FUNCTION_BLOCK FB_Robotersteuerung
VAR_INPUT
    bEnable     : BOOL;
    bExecute    : BOOL;

	bSensBand4 	: BOOL;
	bSensEndX : BOOL;
	bSensEndY : BOOL;
	bSensEndZ : BOOL;
	bSensEndG : BOOL;
END_VAR

VAR_OUTPUT
    eState          : eBetriebszustand;
    bBrakeZ         : BOOL;
    bGripperClosed  : BOOL;
END_VAR

VAR_IN_OUT
    axX : Axis_Ref;
    axY : Axis_Ref;
    axZ : Axis_Ref;
	axG : Axis_Ref;
	
	nLagerIndex : INT; 
END_VAR

VAR
    fbAchseX : FB_AchsenRoboter;
    fbAchseY : FB_AchsenRoboter;
    fbAchseZ : FB_AchsenRoboter;
	fbAchseG : FB_AchsenRoboter;
	
    fbWaage 	: FB_Waage_Temp;
    fbThermo	: FB_Thermo_Temp;

	rGzu 	: REAL 	:= 9.5;
	rGauf 	: REAL 	:= 6.5;
	
    bGreifer	: BOOL;
    nState   	: INT;
END_VAR

fbAchseX(
    bEnable := bEnable,
    bExecute := ,
    rPosition := ,
    bSensEndstop := bSensEndX,
    eState => ,
    ax := axX);

fbAchseY(
    bEnable := bEnable,
    bExecute := ,
    rPosition := ,
    bSensEndstop := bSensEndY,
    eState => ,
    ax := axY);

fbAchseZ(
    bEnable := bEnable,
    bExecute := ,
    rPosition := ,
    bSensEndstop := bSensEndZ,
    eState => ,
    ax := axZ);

fbAchseG(
    bEnable := bEnable,
    bExecute := ,
    rPosition := ,
    bSensEndstop := bSensEndG,
    eState => ,
    ax := axG);

fbWaage();
fbThermo();

CASE nState OF

    0: // OFF
        eState := eBetriebszustand.Off;
        bBrakeZ := FALSE;
        bGripperClosed := FALSE;
		nLagerIndex := 1;
        fbAchseG(bExecute := TRUE, rPosition := rGauf, ax := axG);
        IF bEnable THEN
            nState := 10;
        END_IF

    10: // INIT
        eState := eBetriebszustand.Init;
        bBrakeZ := FALSE;
		fbAchseX(bExecute := TRUE, rPosition := GVL_PosKinematic.pXHome, ax := axX);
        fbAchseY(bExecute := TRUE, rPosition := GVL_PosKinematic.pYHome, ax := axY);
		fbAchseZ(bExecute := TRUE, rPosition := GVL_PosKinematic.pZHome, ax := axZ);
        IF fbAchseX.eState = eBetriebszustand.Done AND fbAchseY.eState = eBetriebszustand.Done AND fbAchseZ.eState = eBetriebszustand.Done THEN
			fbAchseX.bExecute := FALSE;
			fbAchseY.bExecute := FALSE;
			fbAchseZ.bExecute := FALSE;
        	nState := 20;
		END_IF
    20: // READY
        eState := eBetriebszustand.Ready;
        IF bBandSens4 THEN
            nState := 30;
        END_IF

    30: // Z-Achse sicherheits Ebene
        bBrakeZ := TRUE;
        fbAchseZ(bExecute := TRUE, rPosition := GVL_PosKinematic.pZoff, ax := axZ);
        IF fbAchseZ.eState = eBetriebszustand.Done THEN
			fbAchseZ.bExecute := FALSE;
            nState := 31;
        END_IF

    31: // XY Abfüllstation
    IF fbAchseZ.rPosition <= GVL_PosKinematic.pZOff  THEN
		bBrakeZ := FALSE;
        fbAchseX(bExecute := TRUE, rPosition := GVL_PosKinematic.pXconv, ax := axX);
        fbAchseY(bExecute := TRUE, rPosition := GVL_PosKinematic.pYconv, ax := axY);
        IF fbAchseX.eState = eBetriebszustand.Done AND fbAchseY.eState = eBetriebszustand.Done THEN
			fbAchseX.bExecute := FALSE;
			fbAchseY.bExecute := FALSE;
            nState := 32;
        END_IF
    END_IF

    32: // Z-Achse Greifenhöhe
	IF fbAchseX.rPosition = GVL_PosKinematic.pXconv AND 
	   fbAchseY.rPosition = GVL_PosKinematic.pYconv THEN
	   bBrakeZ := TRUE;
        fbAchseZ(bExecute := TRUE, rPosition := GVL_PosKinematic.pZconv, ax := axZ);
        IF fbAchseZ.eState = eBetriebszustand.Done THEN
			fbAchseZ.bExecute := FALSE;
            nState := 33;
        END_IF
	END_IF
	
    33: // Greifen
	IF fbAchseZ.rPosition = GVL_PosKinematic.pZconv AND fbAchseZ.bExecute = FALSE THEN
		bBrakeZ := FALSE;
        fbAchseG(bExecute := TRUE, rPosition := rGzu, ax := axG);
        IF fbAchseG.eState = eBetriebszustand.Done THEN
			fbAchseG.bExecute := FALSE;
            bGripperClosed := TRUE;
            nState := 34;
        END_IF
	END_IF
	
    34: // Z-Achse sicherheits Ebene
	IF fbAchseg.rPosition = rGzu THEN
		bBrakeZ := TRUE;
        fbAchseZ(bExecute := TRUE, rPosition := GVL_PosKinematic.pZoff, ax := axZ);
        IF fbAchseZ.eState = eBetriebszustand.Done THEN
			fbAchseZ.bExecute := FALSE;
            bBrakeZ := TRUE;
            nState := 40;
        END_IF
	END_IF
	
    40: // XY Waage
    IF fbAchseZ.rPosition <= GVL_PosKinematic.pZOff  THEN
		bBrakeZ := FALSE;
        fbAchseX(bExecute := TRUE, rPosition := GVL_PosKinematic.pXscale, ax := axX);
        fbAchseY(bExecute := TRUE, rPosition := GVL_PosKinematic.pYscale, ax := axY);
        IF fbAchseX.eState = eBetriebszustand.Done AND fbAchseY.eState = eBetriebszustand.Done THEN
			fbAchseX.bExecute := FALSE;
			fbAchseY.bExecute := FALSE;
            nState := 41;
        END_IF
    END_IF

    41: // Z-Achse Ablegen
	IF fbAchseX.rPosition = GVL_PosKinematic.pXscale AND 
	   fbAchseY.rPosition = GVL_PosKinematic.pYscale THEN
	    bBrakeZ := TRUE;
        fbAchseZ(bExecute := TRUE, rPosition := GVL_PosKinematic.pZscale, ax := axZ);
        IF fbAchseZ.eState = eBetriebszustand.Done THEN
			fbAchseZ.bExecute := FALSE;
            nState := 42;
        END_IF
	END_IF
	
    42: // Greifer öffnen
	IF fbAchseZ.rPosition = GVL_PosKinematic.pZscale THEN
		bBrakeZ := FALSE;
        fbAchseG(bExecute := TRUE, rPosition := rGauf, ax := axG);
        IF fbAchseG.eState = eBetriebszustand.Done THEN
			fbAchseG.bExecute := FALSE;
            bGripperClosed := FALSE;
            nState := 43;
        END_IF
	END_IF
	
    43: // Waagenprozess
	IF fbAchseG.rPosition = rGauf THEN
        fbWaage(bEnable := TRUE, bExecute := TRUE);
        IF fbWaage.eState = eBetriebszustand.Done THEN
            fbWaage.bExecute := FALSE;
            nState := 44;
        END_IF
	END_IF
	
    44: // Greifen
	IF fbWaage.bExecute = FALSE THEN 
        fbAchseG(bExecute := TRUE, rPosition := rGzu, ax := axG);
        IF fbAchseG.eState = eBetriebszustand.Done THEN
			fbAchseG.bExecute := FALSE;
            bGripperClosed := TRUE;
            nState := 45;
        END_IF
	END_IF
    45: // Z-Achse sicherheits Ebene
	IF fbAchseG.rPosition = rGzu THEN
		bBrakeZ := TRUE;
        fbAchseZ(bExecute := TRUE, rPosition := GVL_PosKinematic.pZoff, ax := axZ);
        IF fbAchseZ.eState = eBetriebszustand.Done THEN
			fbAchseZ.bExecute := FALSE;
            nState := 50;
        END_IF
	END_IF
	
    50: // XY Thermobehandlung
    IF fbAchseZ.rPosition <= GVL_PosKinematic.pZOff  THEN
		bBrakeZ := FALSE;
        fbAchseX(bExecute := TRUE, rPosition := GVL_PosKinematic.pXheat, ax := axX);
        fbAchseY(bExecute := TRUE, rPosition := GVL_PosKinematic.pYheat, ax := axY);
        IF fbAchseX.eState = eBetriebszustand.Done AND fbAchseY.eState = eBetriebszustand.Done THEN
			fbAchseX.bExecute := FALSE;
			fbAchseY.bExecute := FALSE;
            nState := 51;
        END_IF
    END_IF

    51: // Z-Achse ablegen
	IF fbAchseX.rPosition = GVL_PosKinematic.pXheat AND
	   fbAchseY.rPosition = GVL_PosKinematic.pYheat THEN
	    bBrakeZ := TRUE;
        fbAchseZ(bExecute := TRUE, rPosition := GVL_PosKinematic.pZheat, ax := axZ);
        IF fbAchseZ.eState = eBetriebszustand.Done THEN
			fbAchseZ.bExecute := FALSE;
            nState := 52;
        END_IF
	END_IF
	
    52: // Greifer öffnen
	IF fbAchseZ.rPosition = GVL_PosKinematic.pZheat  THEN
		bBrakeZ := FALSE;
        fbAchseG(bExecute := TRUE, rPosition := rGauf, ax := axG);
        IF fbAchseG.eState = eBetriebszustand.Done THEN
			fbAchseG.bExecute := FALSE;
            bGripperClosed := FALSE;
            nState := 53;
        END_IF
	END_IF
	
    53: // Thermobehandlung
	IF fbAchseG.rPosition = rGauf THEN
        fbThermo(bEnable := TRUE, bExecute := TRUE);
        IF fbThermo.eState = eBetriebszustand.Done THEN
            fbThermo.bExecute := FALSE;
            nState := 54;
        END_IF
	END_IF
	
    54: // Greifen
	IF fbTHermo.bExecute = FALSE THEN
    fbAchseG(bExecute := TRUE, rPosition := rGzu, ax := axG);
    IF fbAchseG.eState = eBetriebszustand.Done THEN
		fbAchseG.bExecute := FALSE;
        bGripperClosed := TRUE;
        nState := 55;
    END_IF
	END_IF

    55: // Z-Achse Sicheitsebene
	IF fbAchseG.rPosition = rGzu THEN
		bBrakeZ := TRUE;
        fbAchseZ(bExecute := TRUE, rPosition := GVL_PosKinematic.pZOff, ax := axZ);
        IF fbAchseZ.eState = eBetriebszustand.Done THEN
			fbAchseZ.bExecute := FALSE;
			bBrakeZ := FALSE;
            nState := 60;
        END_IF
	END_IF
	
    60: // XY Lager
	IF fbAchseZ.rPosition <= GVL_PosKinematic.pZoff THEN
		CASE nLagerIndex OF
        1:
            fbAchseX.rPosition := GVL_PosKinematic.pX1stor;
        2:
            fbAchseX.rPosition := GVL_PosKinematic.pX2stor;
        3:
            fbAchseX.rPosition := GVL_PosKinematic.pX3stor;
		4:
			fbAchseX.rPosition := GVL_PosKinematic.pX4stor;
        ELSE
            fbAchseX.rPosition := GVL_PosKinematic.pX1stor;
    	END_CASE
        fbAchseX(bExecute := TRUE, ax := axX);
        fbAchseY(bExecute := TRUE, rPosition := GVL_PosKinematic.pYstor, ax := axY);
        IF fbAchseX.eState = eBetriebszustand.Done AND fbAchseY.eState = eBetriebszustand.Done THEN
          	fbAchseX.bExecute := FALSE;
		    fbAchseY.bExecute := FALSE;
			nState := 61;
        END_IF
	END_IF
	
    61: // Z-Achse ablegen
	IF fbAchseY.rPosition = GVL_PosKinematic.pYstor THEN
	    bBrakeZ := TRUE;
        fbAchseZ(bExecute := TRUE, rPosition := GVL_PosKinematic.pZstor, ax := axZ);
        IF fbAchseZ.eState = eBetriebszustand.Done THEN
			fbAchseZ.bExecute := FALSE;
            nState := 62;
        END_IF
	END_IF
	
    62: // Greifer öffnen
	IF fbAchseZ.rPosition = GVL_PosKinematic.pZstor THEN
		bBrakeZ := FALSE;
        fbAchseG(bExecute := TRUE, rPosition := rGauf, ax := axG);
        IF fbAchseG.eState = eBetriebszustand.Done THEN
			fbAchseG.bExecute := FALSE;
            bGripperClosed := FALSE;
            nState := 70;
        END_IF
	END_IF
	
    70: // Z-Achse sicherheits Ebene
	IF fbAchseG.rPosition = rGauf THEN
		bBrakeZ := TRUE;
        fbAchseZ(bExecute := TRUE, rPosition := GVL_PosKinematic.pZoff, ax := axZ);
        IF fbAchseZ.eState = eBetriebszustand.Done THEN
			fbAchseZ.bExecute := FALSE;
            nState := 71;
        END_IF
	END_IF
	
    71: // XY Home
    IF fbAchseZ.rPosition <= GVL_PosKinematic.pZOff THEN
		bBrakeZ := FALSE;
        fbAchseX(bExecute := TRUE, rPosition := GVL_PosKinematic.pXhome, ax := axX);
        fbAchseY(bExecute := TRUE, rPosition := GVL_PosKinematic.pYhome, ax := axY);
        IF fbAchseX.eState = eBetriebszustand.Done AND fbAchseY.eState = eBetriebszustand.Done THEN
			fbAchseX.bExecute := FALSE;
			fbAchseY.bExecute := FALSE;
            nState := 72;
        END_IF
    END_IF

    72: // Z-Achse senken
	IF fbAchseX.rPosition = GVL_PosKinematic.pXhome AND
	   fbAchseY.rPosition = GVL_PosKinematic.pYhome THEN
	    bBrakeZ := TRUE;
        fbAchseZ(bExecute := TRUE, rPosition := GVL_PosKinematic.pZhome, ax := axZ);
        IF fbAchseZ.eState = eBetriebszustand.Done THEN
			fbAchseZ.bExecute := FALSE;
            bBrakeZ := TRUE;
            nState := 80;
        END_IF
	END_IF
	
    80: // Done
	IF fbAchseZ.rPosition = GVL_PosKinematic.pZhome THEN
		bBrakeZ := FALSE;
        eState := eBetriebszustand.Done;
	
			IF nLagerIndex < 5 THEN
				nLagerIndex := nLagerIndex + 1;
			END_IF
	
			IF NOT bExecute THEN
				nState := 0;
			END_IF
    
        IF NOT bExecute THEN
            nState := 20;
        END_IF
	END_IF
END_CASE

END_FUNCTION_BLOCK

(* stored: Version 1.1.0.1, ProductVersion 3.1.4024.15
   POU FB_Robotersteuerung: Id {58efb2c0-84e8-473e-9583-d46c3f979c12}, SpecialFunc None *)
